// TIA Portal V17 export
// export: Created 2022-07-20T06:59:44.2149616Z, ExportSetting WithDefaults, DisplayName Totally Integrated Automation Portal, DisplayVersion V17, DisplayName TIA Portal Openness, DisplayVersion V17, DisplayName TIA Portal Version Control Interface, DisplayVersion V17, DisplayName SINAMICS Startdrive Advanced, DisplayVersion V17, DisplayName SINAMICS Startdrive G130, G150, S120, S150, SINAMICS MV, S210, DisplayVersion V17, DisplayName SINAMICS Startdrive G110M, G120, G120C, G120D, G120P, G115D, DisplayVersion V17, DisplayName STEP 7 Professional, DisplayVersion V17, DisplayName STEP 7 Safety, DisplayVersion V17, DisplayName WinCC Advanced, DisplayVersion V17
FUNCTION "FC10071_ScalingLamUVErrorCode" : Void   // FC10071, LAD
TITLE = FC10071_ScalingLamUVErrorCode
{ S7_Optimized_Access := 'TRUE' }
AUTHOR : Jonathan
FAMILY : 1007x_DRYER
VERSION : 1.0
// Release note : 
// 1.0 - Feature developped
// stored: AutoNumber false, IsIECCheckEnabled false, SetENOAutomatically false, UDAEnableTagReadback false
   VAR_INPUT
      AnalogValue : Int;
   END_VAR
   VAR_OUTPUT
      VoltageValue : Real;
   END_VAR
BEGIN

REGION Network 1 (SCL)




   CASE #AnalogValue OF
       0..1382:  
           #VoltageValue := 0.0;
       1383..2765:  
           #VoltageValue := 0.5;
       2766..4148 :
           #VoltageValue := 1.0;
       4149..5531 :
           #VoltageValue := 1.5;
       5532..6914 :
           #VoltageValue := 2.0;
       6915..8297 :
           #VoltageValue := 2.5;
       8298..9680 :
           #VoltageValue := 3.0;
       9681..11063 :
           #VoltageValue := 3.5;
       11064..12446 :
           #VoltageValue := 4.0;
       12447..13829 :
           #VoltageValue := 4.5;
       13830..15212 :
           #VoltageValue := 5.0;
       15213..16595 :
           #VoltageValue := 5.5;
       16596..17978 :
           #VoltageValue := 6.0;
       17979..19361 :
           #VoltageValue := 6.5;
       19362..20744 :
           #VoltageValue := 7.0;
       20745..22127 :
           #VoltageValue := 7.5;
       22128..23510 :
           #VoltageValue := 8.0;
       23511..24893 :
           #VoltageValue := 8.5;
       24894..26276 :
           #VoltageValue := 9.0;
       26277..27659 :
           #VoltageValue := 9.5;
       27660..29042 :
           #VoltageValue := 10.0;
       ELSE  // Statement section ELSE
           #VoltageValue := 0.0;
   END_CASE;
END_REGION
END_FUNCTION
